FUNCTION_BLOCK FB_Counter
VAR
END_VAR

METHOD AddTwo : DINT
VAR_INPUT
    In1 : DINT;
    In2 : DINT;
END_VAR
AddTwo := In1 + In2;
END_METHOD

END_FUNCTION_BLOCK

(* stored: Version 1.1.0.1
   POU FB_Counter: Id {012b8ed0-2a5c-4bc2-bd74-056604d88c1c}, SpecialFunc None
   Method AddTwo: Id {2fd73b10-3d6d-4b49-8abc-ef2b87de2173} *)
